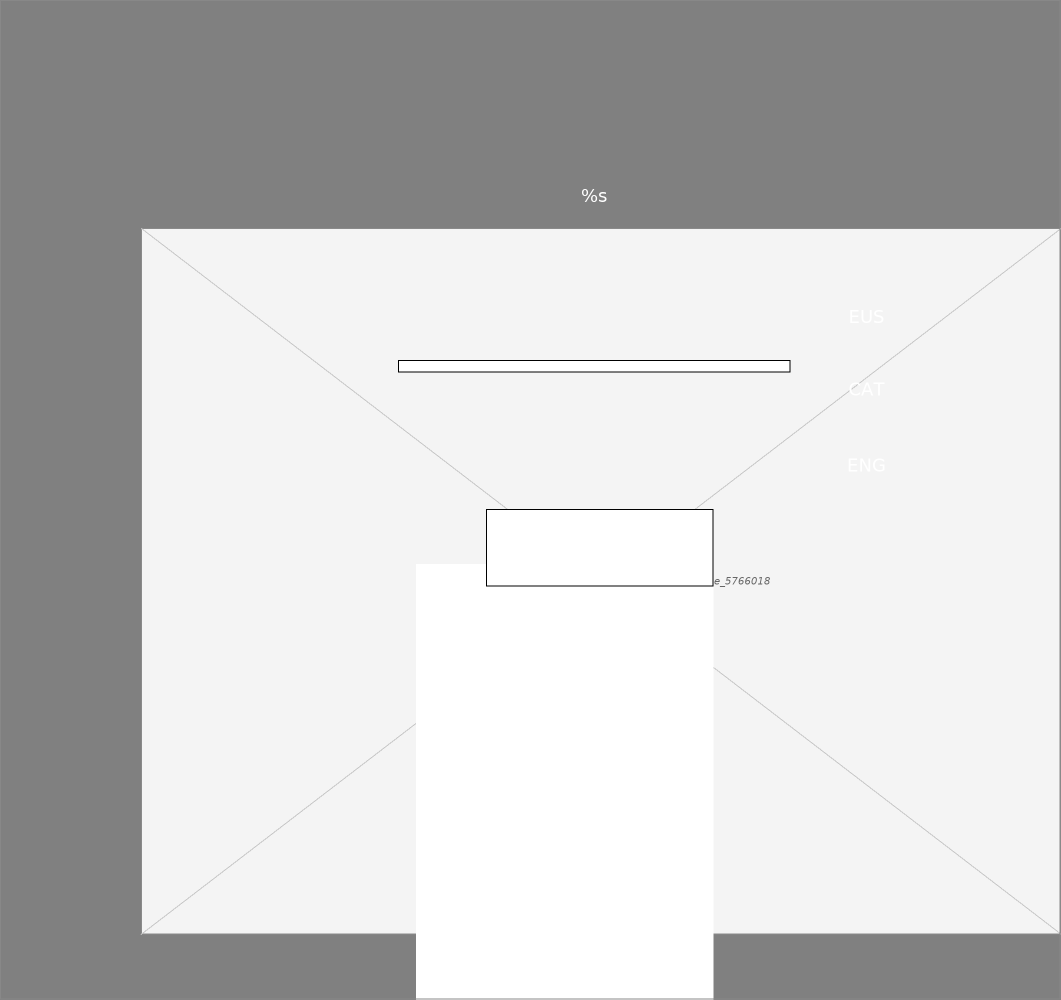
VISUALIZATION disconnected  // 1061x1000
    Image (141,228 920x706), image: ImagePool.pngtree-traffic-lights-clipart-design-png-image_5766018
    Rectangle (398,360 392x12), angle 315
    Rectangle (416,564 297x436)
    RoundedRectangle (486,509 227x77), "ON/OFF"
        toggle MAIN.updateState.HMI_Switch
        OnMouseClick: change screen: mainPage
    RoundedRectangle (424,161 341x70), "%s", text list: 'GlobalTextList', text index: MAIN.mensajeIdioma
    Rectangle (754,287 225x60), "EUS"
        OnMouseClick: ChangeLanguage ChangeLanguage=EUSKERA
        OnMouseClick: execute {
            main.boolCAT := TRUE;
            main.boolENG := TRUE;
            main.boolEUS := FALSE;
        }
    Rectangle (754,357 225x65), "CAT"
        OnMouseClick: ChangeLanguage ChangeLanguage=CATALÀ
        OnMouseClick: execute {
            main.boolCAT := FALSE;
            main.boolENG := TRUE;
            main.boolEUS := TRUE;
        }
    Rectangle (754,436 225x59), "ENG"
        OnMouseClick: ChangeLanguage ChangeLanguage=ENGLISH
        OnMouseClick: execute {
            main.boolCAT := TRUE;
            main.boolENG := FALSE;
            main.boolEUS := TRUE;
        }
END_VISUALIZATION

(* stored: Version 1.1.0.1
   Visu disconnected: Id {3d191336-253b-4049-9c07-50d572e30d01} *)
